E_DALIBridgeCommand.resetDurationTestDoneFlag:
	fbResetDurationTestDoneFlag(
		bStart					:= requestFirstCycle,
		nAddress				:= activeRequest.address,
		eAddressType			:= activeRequest.addressType,
	);
	processResult(
		busy					:= fbResetDurationTestDoneFlag.bBusy,
		bError					:= fbResetDurationTestDoneFlag.bError,
		data					:= 0,
		ipResultMessage			:= fbResetDurationTestDoneFlag.ipResultMessage
	);
	
E_DALIBridgeCommand.resetFunctionTestDoneFlag:
	fbResetFunctionTestDoneFlag(
		bStart					:= requestFirstCycle,
		nAddress				:= activeRequest.address,
		eAddressType			:= activeRequest.addressType,
	);
	processResult(
		busy					:= fbResetFunctionTestDoneFlag.bBusy,
		bError					:= fbResetFunctionTestDoneFlag.bError,
		data					:= 0,
		ipResultMessage			:= fbResetFunctionTestDoneFlag.ipResultMessage
	);
	
E_DALIBridgeCommand.startDurationTest:
	IF emergency THEN
		cancelCommand();
	ELSE
		fbStartDurationTest(
			bStart					:= requestFirstCycle,
			nAddress				:= activeRequest.address,
			eAddressType			:= activeRequest.addressType,
		);
		processResult(
			busy					:= fbStartDurationTest.bBusy,
			bError					:= fbStartDurationTest.bError,
			data					:= 0,
			ipResultMessage			:= fbStartDurationTest.ipResultMessage
		);
	END_IF
	
E_DALIBridgeCommand.startFunctionTest:
	IF emergency THEN
		cancelCommand();
	ELSE
		fbStartFunctionTest(
			bStart					:= requestFirstCycle,
			nAddress				:= activeRequest.address,
			eAddressType			:= activeRequest.addressType,
		);
		processResult(
			busy					:= fbStartFunctionTest.bBusy,
			bError					:= fbStartFunctionTest.bError,
			data					:= 0,
			ipResultMessage			:= fbStartFunctionTest.ipResultMessage
		);
	END_IF
	
E_DALIBridgeCommand.stopTest:
	fbStopTest(
		bStart						:= requestFirstCycle,
		nAddress					:= activeRequest.address,
		eAddressType				:= activeRequest.addressType,
	);
	processResult(
		busy						:= fbStopTest.bBusy,
		bError						:= fbStopTest.bError,
		data						:= 0,
		ipResultMessage				:= fbStopTest.ipResultMessage
	);
	
E_DALIBridgeCommand.setDurationTestInterval:
	fbSetDurationTestInterval(
		bStart						:= requestFirstCycle,
		nAddress					:= activeRequest.address,
		eAddressType				:= activeRequest.addressType,
		nDurationTestInterval		:= activeRequest.data
	);
	processResult(
		busy						:= fbSetDurationTestInterval.bBusy,
		bError						:= fbSetDurationTestInterval.bError,
		data						:= 0,
		ipResultMessage				:= fbSetDurationTestInterval.ipResultMessage
	);
	
E_DALIBridgeCommand.setFunctionTestInterval:
	fbSetFunctionTestInterval(
		bStart						:= requestFirstCycle,
		nAddress					:= activeRequest.address,
		eAddressType				:= activeRequest.addressType,
		nFunctionTestInterval		:= activeRequest.data
	);
	processResult(
		busy						:= fbSetFunctionTestInterval.bBusy,
		bError						:= fbSetFunctionTestInterval.bError,
		data						:= 0,
		ipResultMessage				:= fbSetFunctionTestInterval.ipResultMessage
	);
	
E_DALIBridgeCommand.startIdentification202:
	fbStartIdentification202(
		bStart						:= requestFirstCycle,
		nAddress					:= activeRequest.address,
		eAddressType				:= activeRequest.addressType,
	);
	processResult(
		busy						:= fbStartIdentification202.bBusy,
		bError						:= fbStartIdentification202.bError,
		data						:= 0,
		ipResultMessage				:= fbStartIdentification202.ipResultMessage
	);
	
E_DALIBridgeCommand.queryGroups:
	fbQueryGroups(
		bStart						:= requestFirstCycle,
		nAddress 					:= activeRequest.address,
		eAddressType				:= activeRequest.addressType
	);
	processResult(
		busy						:= fbQueryGroups.bBusy,
		bError						:= fbQueryGroups.bError,
		data						:= fbQueryGroups.nGroups,
		ipResultMessage				:= fbQueryGroups.ipResultMessage
	);
	
E_DALIBridgeCommand.addToGroup:
	fbAddToGroup(
		bStart 						:= requestFirstCycle,
		nAddress 					:= activeRequest.address,
		eAddressType				:= activeRequest.addressType,
		nGroup						:= activeRequest.data
	);
	processResult(
		busy						:= fbAddToGroup.bBusy,
		bError						:= fbAddToGroup.bError,
		data						:= 0,
		ipResultMessage				:= fbAddToGroup.ipResultMessage
	);
	
E_DALIBridgeCommand.removeFromGroup:
	fbRemoveFromGroup(
		bStart						:= requestFirstCycle,
		nAddress 					:= activeRequest.address,
		eAddressType 				:= activeRequest.addressType,
		nGroup						:= activeRequest.data
	);
	processResult(
		busy						:= fbRemoveFromGroup.bBusy,
		bError						:= fbRemoveFromGroup.bError,
		data						:= 0,
		ipResultMessage				:= fbRemoveFromGroup.ipResultMessage
	);
	
E_DALIBridgeCommand.testCommand:
	processResult(
		busy := FALSE,
		data := 123,
		bError := FALSE,
		ipResultMessage := NULL
	);

ELSE
	activeRequest.command := E_DALIBridgeCommand.idle;
END_CASE

processNotifications();

requestFirstCycle := FALSE;

METHOD PRIVATE cancelCommand
VAR_INPUT
END_VAR

VAR
	tmpResponse: ST_DALIBridgeResponse;
END_VAR
// generate response
tmpResponse.valid := TRUE;
tmpResponse.data := 0;
tmpResponse.error := TRUE;
tmpResponse.message := 'Emergency in progress';
tmpResponse.sequence := THIS^.activeRequestSequence;

// return to the idle state, ready for a new request
THIS^.activeRequest.command := E_DALIBridgeCommand.idle;
// publish the response
THIS^.rpcResponse := tmpResponse;
END_METHOD

METHOD FB_init : BOOL
VAR_INPUT
	bInitRetains : BOOL; // if TRUE, the retain variables are initialized (warm start / cold start)
	bInCopyCode : BOOL;  // if TRUE, the instance afterwards gets moved into the copy code (online change)
	
	communication : I_DALICommunication;
END_VAR
THIS^.communication := communication;
END_METHOD

METHOD PRIVATE initCommunication
VAR_INPUT
END_VAR
VAR
	i : INT;
END_VAR
IF communication = 0 THEN
	RETURN;
END_IF

FOR i := 0 TO GVL_DALIBridge.maxInputEventListeners-1 DO
	fbsGetInputNotification[i].ipDALICommunication := communication;
END_FOR

fbEmergencyPowerOn.ipDALICommunication 		:= communication;
fbDirectArcPowerControl.ipDALICommunication := communication;
fbQueryActualLevel.ipDALICommunication 		:= communication;
fbQueryStatus.ipDALICommunication 			:= communication;
fbSetEventScheme.ipDALICommunication 		:= communication;
fbQueryEventScheme.ipDALICommunication 		:= communication;
fbSetEventFilter.ipDALICommunication 		:= communication;
fbQueryEventFilter.ipDALICommunication 		:= communication;
fbIdentifyDevice102.ipDALICommunication 	:= communication;
fbIdentifyDevice103.ipDALICommunication 	:= communication;
fbEnableInstance.ipDALICommunication 		:= communication;
fbGoToScene.ipDALICommunication 			:= communication;
fbSetFadeTime.ipDALICommunication 			:= communication;
fbQueryInputValue.ipDALICommunication		:= communication;

fbQueryBatteryCharge.ipDALICommunication    	:= communication;
fbQueryDurationTestResult.ipDALICommunication 	:= communication;
fbQueryEmergencyMode.ipDALICommunication        := communication;
fbQueryEmergencyStatus.ipDALICommunication  	:= communication;
fbQueryFailureStatus.ipDALICommunication		:= communication;
fbQueryRatedDuration.ipDALICommunication		:= communication;
fbQueryTestTiming.ipDALICommunication			:= communication;
fbResetDurationTestDoneFlag.ipDALICommunication := communication;
fbResetFunctionTestDoneFlag.ipDALICommunication := communication;
fbStartDurationTest.ipDALICommunication 		:= communication;
fbStartFunctionTest.ipDALICommunication 		:= communication;
fbStopTest.ipDALICommunication					:= communication;
fbSetDurationTestInterval.ipDALICommunication   := communication;
fbSetFunctionTestInterval.ipDALICommunication   := communication;
fbStartIdentification202.ipDALICommunication    := communication;
END_METHOD

METHOD PRIVATE isFirstCycle : BOOL
VAR_INPUT
END_VAR
VAR_INST
	fbGetCurTaskIndex : GETCURTASKINDEX;
END_VAR
fbGetCurTaskIndex();
isFirstCycle := TwinCAT_SystemInfoVarList._TaskInfo[fbGetCurTaskIndex.index].FirstCycle;
END_METHOD

METHOD PRIVATE processNotifications : BOOL
VAR_INPUT
END_VAR
VAR
	i 				: DINT;
	eventsProcessed : BYTE := 0;
	
	currentParams   : REFERENCE TO ST_DALIBridgeInputEventParams;
	currentFb 		: REFERENCE TO FB_DALIGetInputNotification;
	currentEvent    : REFERENCE TO ST_DALIBridgeInputEvent;
	
	newNotif : ST_DALIBridgeNotification;
END_VAR
IF NOT notificationAcked THEN
	// cannot process more notifications until the current notification has been ACKed
	processNotifications := FALSE;
	RETURN;
END_IF

newNotif.valid := FALSE;

// for every active notification listener
FOR i := 0 TO numInputEventListeners-1 DO
	IF (eventsProcessed >= GVL_DALIBridge.maxInputEventsPerNotification) THEN
		// stop processing if the event buffer is full
		EXIT;
	END_IF	

	currentFb REF= fbsGetInputNotification[i];
	currentParams REF= inputEventListenerParams[i];
	
	// check for a new event
	currentFb(
		bEnable := TRUE,
		eEventScheme := currentParams.eventScheme,
		nAddressInfo1 := currentParams.addressInfo1,
		nAddressInfo2 := currentParams.addressInfo2
	);
	
	// don't add to event array if no new data was found
	IF NOT currentFb.bNewData THEN
		CONTINUE;
	END_IF
	
	// populate the event entry
	currentEvent REF= newNotif.inputEvents[eventsProcessed];
	currentEvent.data := currentFb.nEventInfo;
	currentEvent.error := currentFb.bError;
	currentFb.ipResultMessage.RequestEventText(
		nLangId := 1033,
		sResult := currentEvent.message,
		nResultSize := SIZEOF(currentEvent.message)
	);
	currentEvent.parameters := inputEventListenerParams[i];
	currentEvent.status := currentFb.ipResultMessage.nEventId;
	
	eventsProcessed := eventsProcessed + 1;
END_FOR

IF (eventsProcessed > 0) THEN
	newNotif.sequence := notificationCounter;
	notificationCounter := notificationCounter + 1;
	newNotif.nInputEvents := eventsProcessed;
	newNotif.valid := TRUE;
	
	notification := newNotif;
	notificationAcked := FALSE;
END_IF
END_METHOD

METHOD PRIVATE processResult
VAR_INPUT
	busy 			: BOOL;
	data            : LWORD;
	bError 			: BOOL;
	ipResultMessage	: Tc3_EventLogger.I_TcMessage;
END_VAR
VAR
	tmpResponse: ST_DALIBridgeResponse;
END_VAR
IF (busy) THEN
	// continue executing the command function block until it is no longer busy
	RETURN;
END_IF

// generate response
tmpResponse.valid := TRUE;
tmpResponse.data := data;
tmpResponse.error := bError;
tmpResponse.sequence := THIS^.activeRequestSequence;
IF ipResultMessage = 0 THEN
	ADSLOGSTR(
		msgCtrlMask := ADSLOG_MSGTYPE_WARN,
		msgFmtStr := 'FB_DALIBridge.processResult: ipResultMessage is null',
		strArg := ''
	);
	tmpResponse.status := 0;
	tmpResponse.message := 'ipResultMessage NULL';
ELSE
	tmpResponse.status := ipResultMessage.nEventId;
	ipResultMessage.RequestEventText(1033, tmpResponse.message, SIZEOF(tmpResponse.message));
END_IF

// return to the idle state, ready for a new request
THIS^.activeRequest.command := E_DALIBridgeCommand.idle;
// publish the response
THIS^.rpcResponse := tmpResponse;
END_METHOD

{attribute 'TcRpcEnable' := '1'}
METHOD PUBLIC RpcAckNotification : BOOL
VAR_INPUT
	// The notification sequence number to acknowledge
	sequence : ULINT;
END_VAR
IF notificationAcked THEN
	// can't acknowledge a notification twice
	RpcAckNotification := FALSE;
	RETURN;
END_IF

IF sequence <> notification.sequence THEN
	// attempt to acknowledge a notification with the wrong sequence number
	RpcAckNotification := FALSE;
	RETURN;
END_IF

RpcAckNotification := TRUE;
notificationAcked := TRUE;
END_METHOD

{attribute 'TcRpcEnable' := '1'}
METHOD PUBLIC RpcAddInputEventListener : BOOL
VAR_INPUT
	parameters : ST_DALIBridgeInputEventParams;
END_VAR
VAR
	i : INT;
END_VAR
ADSLOGSTR(
		msgFmtStr := 'add event listener',
		strArg := '',
		msgCtrlMask := ADSLOG_MSGTYPE_LOG
);

FOR i := 0 TO numInputEventListeners-1 DO
	IF (parameters.eventScheme = inputEventListenerParams[i].eventScheme
		AND parameters.addressInfo1 = inputEventListenerParams[i].addressInfo1
		AND parameters.addressInfo2 = inputEventListenerParams[i].addressInfo2) 
	THEN
		// the desired event listener is already enabled
		RpcAddInputEventListener := TRUE;
		RETURN;
	END_IF
END_FOR

IF numInputEventListeners >= GVL_DALIBridge.maxInputEventListeners THEN
	// notification listeners are full
	RpcAddInputEventListener := FALSE;
	RETURN;
END_IF

inputEventListenerParams[numInputEventListeners] := parameters;
numInputEventListeners := numInputEventListeners + 1;

RpcAddInputEventListener := TRUE;
END_METHOD

{attribute 'TcRpcEnable' := '1'}
METHOD PUBLIC RpcHandshake
VAR_INPUT
END_VAR
VAR_OUTPUT
	protocolVersion : INT;
END_VAR
protocolVersion := 2;
END_METHOD

(* Called by an external API consumer over RPC to start a DALI request.
   Returns TRUE if the request was accepted. If the bridge is busy, then this returns FALSE
   and the request will not be processed. *)
{attribute 'TcRpcEnable' := '1'}
METHOD PUBLIC RpcRequest : BOOL
VAR_INPUT
	// The DALI operation that the caller wants the DALI Bridge to perform.
	request : ST_DALIBridgeRequest;
END_VAR
VAR_OUTPUT
	// A sequence number that will allow the caller to identify the response value.
	sequence : ULINT;
END_VAR
// reject request if bridge is busy processing a previous request
IF (THIS^.activeRequest.command <> E_DALIBridgeCommand.idle) THEN
	RpcRequest := FALSE;
	RETURN;
END_IF

// save the request, so it will begin processing next cycle
THIS^.activeRequest := request;
THIS^.activeRequestSequence := THIS^.requestCounter;
sequence := THIS^.activeRequestSequence;

// advance sequence counter
THIS^.requestCounter := THIS^.requestCounter + 1;

// The next cycle will be the first cycle of the new request
THIS^.requestFirstCycle := TRUE;

RpcRequest := TRUE;
END_METHOD

{attribute 'TcRpcEnable' := '1'}
METHOD PUBLIC RpcReset
VAR_INPUT
END_VAR
numInputEventListeners := 0;
notificationAcked := TRUE;
activeRequest.command := E_DALIBridgeCommand.idle;
ADSLOGSTR(
		msgFmtStr := 'reset FB_DALIBridge',
		strArg := '',
		msgCtrlMask := ADSLOG_MSGTYPE_LOG
);
END_METHOD

END_FUNCTION_BLOCK

// ---- GlobalTextList.TcGTLO
TEXTLIST GlobalTextList
  621 = '%d'
  665 = '%d %'
  2025 = '%d ms'
  1540 = '%d s'
  646 = '%s'
  640 = '0'
  641 = '1'
  661 = '10'
  662 = '11'
  663 = '12'
  999 = '13'
  1000 = '14'
  1001 = '15'
  1002 = '16'
  1003 = '17'
  1004 = '18'
  1005 = '19'
  642 = '2'
  1006 = '20'
  1007 = '21'
  1008 = '22'
  1009 = '23'
  1010 = '24'
  1011 = '25'
  1012 = '26'
  1013 = '27'
  1014 = '28'
  1015 = '29'
  654 = '3'
  1016 = '30'
  1017 = '31'
  1018 = '32'
  1019 = '33'
  1020 = '34'
  1021 = '35'
  1022 = '36'
  1023 = '37'
  1024 = '38'
  1025 = '39'
  655 = '4'
  1026 = '40'
  1027 = '41'
  1028 = '42'
  1029 = '43'
  1030 = '44'
  1031 = '45'
  1032 = '46'
  1033 = '47'
  1034 = '48'
  1035 = '49'
  656 = '5'
  358 = '50'
  359 = '51'
  360 = '52'
  361 = '53'
  362 = '54'
  363 = '55'
  364 = '56'
  365 = '57'
  366 = '58'
  367 = '59'
  657 = '6'
  368 = '60'
  369 = '61'
  370 = '62'
  371 = '63'
  658 = '7'
  659 = '8'
  660 = '9'
  1089 = 'AC-supply possible'
  644 = 'Actual Level:'
  650 = 'Address Type'
  1175 = 'AM Operation active:'
  1044 = 'AM operation possible'
  2131 = 'Back'
  2471 = 'Bit 0'
  379 = 'Bit 1'
  2734 = 'Bit 2'
  2320 = 'Bit 3'
  929 = 'Bit 4'
  2576 = 'Bit 5'
  2065 = 'Bit 6'
  1623 = 'Bit 7'
  626 = 'Broadcast'
  515 = 'Button pressed'
  498 = 'Button released'
  527 = 'Button stuck / free'
  593 = 'Cancel Hold Timer'
  2101 = 'Catch Movement'
  2319 = 'Catching:'
  897 = 'Change Addresses'
  372 = 'Choose group:'
  98 = 'Choose scene:'
  618 = 'Complete new installation \n(all addresses will be removed)'
  807 = 'Control'
  645 = 'Control Gear Failure:'
  146 = 'Control LED'
  445 = 'Current protection active:'
  1716 = 'Current protection device'
  668 = 'Current protection enabled:'
  5 = 'Current Protector Enabled '
  1902 = 'DALI Line:'
  1135 = 'DC-supply possible'
  560 = 'Deadtime Timer:'
  1180 = 'DI1 falling edge'
  1218 = 'DI1 rising edge'
  1726 = 'DI2 falling edge'
  1876 = 'DI2 rising edge'
  936 = 'Dimming Curve:'
  2135 = 'Do not lock process image in case of \nDALI commands from DI1 or DI2'
  519 = 'Double press'
  1112 = 'Double Timer Min:'
  482 = 'Double Timer:'
  811 = 'Down'
  486 = 'Enable'
  828 = 'Enable:'
  1982 = 'EventPriority'
  32 = 'EventPriority:'
  1925 = 'EventScheme'
  1113 = 'EventScheme:'
  1841 = 'Extended Fade Time only valid if Fade Time equals 0!'
  310 = 'Extended Version Number'
  649 = 'Fade Running:'
  494 = 'FadeRate'
  499 = 'FadeTime'
  319 = 'Fast Fade Time:'
  1808 = 'Features LED'
  1434 = 'GearType LED'
  815 = 'Go to Scene'
  99 = 'Go to scene'
  625 = 'Group Address'
  568 = 'Hold Timer:'
  311 = 'Hysteresis Min:'
  313 = 'Hysteresis:'
  1117 = 'Identify'
  315 = 'Illuminance Level'
  540 = 'Input Value:'
  544 = 'Instance Error:'
  1038 = 'Instance Number:'
  492 = 'Internal DALI power supply disabled'
  1771 = 'K-Bus Watchdog'
  647 = 'Lamp Failure:'
  506 = 'LED module integrated'
  306 = 'Load Decrease:'
  1137 = 'Load Increase:'
  1811 = 'Lockable bytes: changeable if "Offset 2" has the Value 85 (0x55).\nFor changing use decimal value.'
  1077 = 'Login'
  1294 = 'Logout'
  523 = 'Long press repeat'
  507 = 'Long press start'
  511 = 'Long press stop'
  2046 = 'Memory Bank:'
  584 = 'Movement'
  531 = 'na'
  680 = 'Name'
  926 = 'Name of byte in memory bank'
  56 = 'NewAddress'
  588 = 'No Movement'
  2294 = 'None'
  572 = 'Occupied'
  808 = 'Off'
  674 = 'Offset'
  1329 = 'Offset in memory bank'
  55 = 'OldAddress'
  816 = 'On and Step Up'
  277 = 'Open Circuit:'
  1714 = 'Operator'
  619 = 'Optical feedback'
  963 = 'Output is current controlled'
  826 = 'Output regulated by current:'
  1900 = 'Parameters'
  2547 = 'Parameters Absolute Input Device'
  1580 = 'Parameters Generic Instance'
  309 = 'Parameters Light Sensor'
  556 = 'Parameters Occupancy Sensor'
  465 = 'Parameters Pushbutton Sensor'
  1847 = 'Physical selection supported'
  1071 = 'Please check if Current Protector is present \nby reading parameters first.'
  308 = 'Please select the desired Short Address in the table above.'
  751 = 'Position Event'
  930 = 'Possible Operating Modes LED'
  719 = 'Power pulse operation'
  1744 = 'Power supply integrated'
  1561 = 'PP Operation active:'
  970 = 'PWM Operation active:'
  1882 = 'PWM operation possible'
  1487 = 'Query idle time detection \nenabled'
  701 = 'Query load decrease enabled'
  1351 = 'Query load increase enabled'
  837 = 'Query reduction luminous flux \nregarding thermal overload'
  463 = 'Query short circuit enabled'
  1293 = 'Query thermal switch enabled'
  617 = 'Random Addressing'
  373 = 'Read'
  181 = 'Read Parameters'
  1531 = 'Reads all Fading Parameters'
  810 = 'Recall Max Level'
  809 = 'Recall Min Level'
  186 = 'Ref. Measurement failed:'
  439 = 'Reference System Power'
  580 = 'Repeat'
  470 = 'Repeat Timer:'
  564 = 'Report Timer:'
  2418 = 'Reset inactive process image'
  648 = 'Reset State:'
  1037 = 'Resolution:'
  616 = 'Scan devices by address'
  1036 = 'Scene Level'
  814 = 'Scene:'
  1366 = 'Set Extended Fade Time'
  252 = 'Set Fade Rate'
  1875 = 'Set Fade Time'
  624 = 'Short Address'
  302 = 'Short Address Range'
  1041 = 'Short Address:'
  34 = 'Short Circuit:'
  503 = 'Short press'
  1516 = 'Short Timer Min:'
  478 = 'Short Timer:'
  300 = 'Single Short Address'
  615 = 'Start'
  620 = 'Start with address:'
  643 = 'Status'
  958 = 'Status Absolute Input Device'
  2506 = 'Status Generic Instance'
  82 = 'Status LED'
  317 = 'Status Light Sensor'
  597 = 'Status Occupancy Sensor'
  536 = 'Status Pushbutton Sensor'
  812 = 'Step Down'
  813 = 'Step Down and Off'
  818 = 'Step Up'
  164 = 'Stuck Timer:'
  376 = 'Switch Off'
  375 = 'Switch On'
  2458 = 'Terminal Event'
  1108 = 'Thermal Overload:'
  355 = 'Thermal Shut Down:'
  305 = 'To'
  627 = 'Unaddressed'
  817 = 'Up'
  2521 = 'V%s'
  576 = 'Vacant'
  1205 = 'Value'
  686 = 'Value Dec'
  1435 = 'Value decimal'
  692 = 'Value Hex'
  2231 = 'Value hexadecimal,\nto change use\nvalue decimal'
  374 = 'Write'
  1047 = 'Write default values'
  490 = 'Write parameters'
END_TEXTLIST

// ---- Tc3_DALI_PLC_Commissioning_Tool/GlobalTextList_1.TcGTLO
TEXTLIST GlobalTextList_1
  621 = '%d'
  665 = '%d %'
  2025 = '%d ms'
  1540 = '%d s'
  646 = '%s'
  640 = '0'
  641 = '1'
  661 = '10'
  662 = '11'
  663 = '12'
  999 = '13'
  1000 = '14'
  1001 = '15'
  1002 = '16'
  1003 = '17'
  1004 = '18'
  1005 = '19'
  642 = '2'
  1006 = '20'
  1007 = '21'
  1008 = '22'
  1009 = '23'
  1010 = '24'
  1011 = '25'
  1012 = '26'
  1013 = '27'
  1014 = '28'
  1015 = '29'
  654 = '3'
  1016 = '30'
  1017 = '31'
  1018 = '32'
  1019 = '33'
  1020 = '34'
  1021 = '35'
  1022 = '36'
  1023 = '37'
  1024 = '38'
  1025 = '39'
  655 = '4'
  1026 = '40'
  1027 = '41'
  1028 = '42'
  1029 = '43'
  1030 = '44'
  1031 = '45'
  1032 = '46'
  1033 = '47'
  1034 = '48'
  1035 = '49'
  656 = '5'
  358 = '50'
  359 = '51'
  360 = '52'
  361 = '53'
  362 = '54'
  363 = '55'
  364 = '56'
  365 = '57'
  366 = '58'
  367 = '59'
  657 = '6'
  368 = '60'
  369 = '61'
  370 = '62'
  371 = '63'
  658 = '7'
  659 = '8'
  660 = '9'
  1089 = 'AC-supply possible'
  644 = 'Actual Level:'
  650 = 'Address Type'
  1175 = 'AM Operation active:'
  1044 = 'AM operation possible'
  2131 = 'Back'
  2471 = 'Bit 0'
  379 = 'Bit 1'
  2734 = 'Bit 2'
  2320 = 'Bit 3'
  929 = 'Bit 4'
  2576 = 'Bit 5'
  2065 = 'Bit 6'
  1623 = 'Bit 7'
  803 = 'Broadcast'
  515 = 'Button pressed'
  498 = 'Button released'
  527 = 'Button stuck / free'
  593 = 'Cancel Hold Timer'
  2101 = 'Catch Movement'
  2319 = 'Catching:'
  897 = 'Change Addresses'
  372 = 'Choose group:'
  98 = 'Choose scene:'
  618 = 'Complete new installation \n(all addresses will be removed)'
  807 = 'Control'
  645 = 'Control Gear Failure:'
  146 = 'Control LED'
  445 = 'Current protection active:'
  1716 = 'Current protection device'
  668 = 'Current protection enabled:'
  5 = 'Current Protector Enabled '
  1902 = 'DALI Line:'
  334 = 'DALI Power Supply'
  1135 = 'DC-supply possible'
  560 = 'Deadtime Timer:'
  1180 = 'DI1 falling edge'
  1218 = 'DI1 rising edge'
  1726 = 'DI2 falling edge'
  1876 = 'DI2 rising edge'
  936 = 'Dimming Curve:'
  169 = 'Do not lock process image'
  2135 = 'Do not lock process image in case of \nDALI commands from DI1 or DI2'
  2344 = 'Do not lock process image in case of DALI commands from DI1 or DI2'
  519 = 'Double press'
  1112 = 'Double Timer Min:'
  482 = 'Double Timer:'
  811 = 'Down'
  486 = 'Enable'
  828 = 'Enable:'
  1982 = 'EventPriority'
  32 = 'EventPriority:'
  494 = 'EventScheme'
  1113 = 'EventScheme:'
  1841 = 'Extended Fade Time only valid if Fade Time equals 0!'
  310 = 'Extended Version Number'
  649 = 'Fade Running:'
  1150 = 'FadeRate'
  1160 = 'FadeTime'
  319 = 'Fast Fade Time:'
  1808 = 'Features LED'
  1434 = 'GearType LED'
  815 = 'Go to Scene'
  99 = 'Go to scene'
  802 = 'Group Address'
  1923 = 'Hier noch die Abfrage der extended version Number\nmit reinbringen, damit klar wird welcher Edition das Gerät angehört.'
  568 = 'Hold Timer:'
  311 = 'Hysteresis Min:'
  313 = 'Hysteresis:'
  1117 = 'Identify'
  2159 = 'Identify 202'
  315 = 'Illuminance Level'
  540 = 'Input Value:'
  544 = 'Instance Error:'
  1038 = 'Instance Number:'
  1374 = 'InstanceType0'
  652 = 'InstanceType1'
  653 = 'InstanceType3'
  664 = 'InstanceType4'
  492 = 'Internal DALI power supply disabled'
  1820 = 'IT0 (Generic Input)'
  1151 = 'IT1 (PushButton)'
  906 = 'IT2 (absolute Input)'
  909 = 'IT2 (Absolute Input)'
  819 = 'IT3 (Occupancy)'
  224 = 'IT4 (Light Sensor)'
  1771 = 'K-Bus Watchdog'
  647 = 'Lamp Failure:'
  506 = 'LED module integrated'
  306 = 'Load Decrease:'
  1137 = 'Load Increase:'
  1811 = 'Lockable bytes: changeable if "Offset 2" has the Value 85 (0x55).\nFor changing use decimal value.'
  523 = 'Long press repeat'
  507 = 'Long press start'
  511 = 'Long press stop'
  2046 = 'Memory Bank:'
  584 = 'Movement'
  531 = 'na'
  842 = 'Name'
  926 = 'Name of byte in memory bank'
  193 = 'NewAddress'
  588 = 'No Movement'
  572 = 'Occupied'
  808 = 'Off'
  835 = 'Offset'
  1329 = 'Offset in memory bank'
  192 = 'OldAddress'
  816 = 'On and Step Up'
  277 = 'Open Circuit:'
  651 = 'OperatingMode'
  619 = 'Optical feedback'
  963 = 'Output is current controlled'
  826 = 'Output regulated by current:'
  1900 = 'Parameters'
  2547 = 'Parameters Absolute Input Device'
  1580 = 'Parameters Generic Instance'
  309 = 'Parameters Light Sensor'
  556 = 'Parameters Occupancy Sensor'
  465 = 'Parameters Pushbutton Sensor'
  1847 = 'Physical selection supported'
  1071 = 'Please check if Current Protector is present \nby reading parameters first.'
  308 = 'Please select the desired Short Address in the table above.'
  751 = 'Position Event'
  930 = 'Possible Operating Modes LED'
  719 = 'Power pulse operation'
  1744 = 'Power supply integrated'
  1561 = 'PP Operation active:'
  970 = 'PWM Operation active:'
  1882 = 'PWM operation possible'
  1487 = 'Query idle time detection \nenabled'
  701 = 'Query load decrease enabled'
  1351 = 'Query load increase enabled'
  837 = 'Query reduction luminous flux \nregarding thermal overload'
  463 = 'Query short circuit enabled'
  1293 = 'Query thermal switch enabled'
  617 = 'Random Addressing'
  373 = 'Read'
  316 = 'Read parameters'
  181 = 'Read Parameters'
  1531 = 'Reads all Fading Parameters'
  810 = 'Recall Max Level'
  809 = 'Recall Min Level'
  186 = 'Ref. Measurement failed:'
  439 = 'Reference System Power'
  580 = 'Repeat'
  470 = 'Repeat Timer:'
  564 = 'Report Timer:'
  2418 = 'Reset inactive process image'
  648 = 'Reset State:'
  1037 = 'Resolution:'
  616 = 'Scan devices by address'
  1036 = 'Scene Level'
  814 = 'Scene:'
  1366 = 'Set Extended Fade Time'
  252 = 'Set Fade Rate'
  1875 = 'Set Fade Time'
  801 = 'Short Address'
  1179 = 'Short Address Range'
  1041 = 'Short Address:'
  34 = 'Short Circuit:'
  503 = 'Short press'
  1516 = 'Short Timer Min:'
  478 = 'Short Timer:'
  1170 = 'Single Short Address'
  615 = 'Start'
  620 = 'Start with address:'
  643 = 'Status'
  958 = 'Status Absolute Input Device'
  2506 = 'Status Generic Instance'
  82 = 'Status LED'
  317 = 'Status Light Sensor'
  597 = 'Status Occupancy Sensor'
  536 = 'Status Pushbutton Sensor'
  812 = 'Step Down'
  813 = 'Step Down and Off'
  818 = 'Step Up'
  164 = 'Stuck Timer:'
  376 = 'Switch Off'
  375 = 'Switch On'
  2458 = 'Terminal Event'
  1108 = 'Thermal Overload:'
  355 = 'Thermal Shut Down:'
  305 = 'To'
  804 = 'Unaddressed'
  817 = 'Up'
  2521 = 'V%s'
  298 = 'V3.1.1.0'
  858 = 'V3.4.0.0'
  395 = 'V3.4.0.1'
  1169 = 'V3.5.0.0'
  576 = 'Vacant'
  1205 = 'Value'
  850 = 'Value Dec'
  1435 = 'Value decimal'
  857 = 'Value Hex'
  2231 = 'Value hexadecimal,\nto change use\nvalue decimal'
  374 = 'Write'
  1047 = 'Write default values'
  490 = 'Write parameters'
END_TEXTLIST

// ---- Tc3_DALI_PLC_Commissioning_Tool/VISUs/TextLists/CommandOnTerminalEvent.TcTLO
TEXTLIST CommandOnTerminalEvent
  0 = 'Do Nothing'
  1 = 'Off'
  2 = 'RecallMaxLevel'
  3 = 'RecallMinLevel'
  4 = 'GoToScene0'
  5 = 'GoToScene1'
  6 = 'GoToScene2'
  7 = 'GoToScene3'
  8 = 'GoToScene4'
  9 = 'GoToScene5'
  10 = 'GoToScene6'
  11 = 'GoToScene7'
  12 = 'GoToScene8'
  13 = 'GoToScene9'
  14 = 'GoToScene10'
  15 = 'GoToScene11'
  16 = 'GoToScene12'
  17 = 'GoToScene13'
  18 = 'GoToScene14'
  19 = 'GoToScene15'
   = ''
END_TEXTLIST

// ---- Tc3_DALI_PLC_Commissioning_Tool/VISUs/TextLists/DimmingCurve.TcTLO
TEXTLIST DimmingCurve
  0 = 'Logarithmic'
  1 = 'Linear'
  255 = 'Unknown'
   = ''
END_TEXTLIST

// ---- Tc3_DALI_PLC_Commissioning_Tool/VISUs/TextLists/EventPriority.TcTLO
TEXTLIST EventPriority
  2 = 'MiddleHigh'
  3 = 'Middle'
  4 = 'MiddleLow'
  5 = 'Low'
  255 = 'Unknown'
   = ''
END_TEXTLIST

// ---- Tc3_DALI_PLC_Commissioning_Tool/VISUs/TextLists/EventScheme.TcTLO
TEXTLIST EventScheme
  0 = '0 - Instance type and number'
  1 = '1 - Short address and instance type'
  2 = '2 - Short address and instance number'
  3 = '3 - Device group and instance type'
  4 = '4 - Instance group and instance type'
   = ''
END_TEXTLIST

// ---- Tc3_DALI_PLC_Commissioning_Tool/VISUs/TextLists/ExtendedFadeTime.TcTLO
TEXTLIST ExtendedFadeTime
  0 = 'No Fade'
  1 = '1 * 100 ms = 100 ms'
  2 = '2 * 100 ms = 200 ms'
  3 = '3 * 100 ms = 300 ms'
  4 = '4 * 100 ms = 400 ms'
  5 = '5 * 100 ms = 500 ms'
  6 = '6 * 100 ms = 600 ms'
  7 = '7 * 100 ms = 700 ms'
  8 = '8 * 100 ms = 800 ms'
  9 = '9 * 100 ms = 900 ms'
  10 = '10 * 100 ms = 1000 ms'
  11 = '11 * 100 ms = 1100 ms'
  12 = '12 * 100 ms = 1200 ms'
  13 = '13 * 100 ms = 1300 ms'
  14 = '14 * 100 ms = 1400 ms'
  15 = '15 * 100 ms = 1500 ms'
  16 = '16 * 100 ms = 1600 ms'
  17 = '1 * 1 s = 1 s'
  18 = '2 * 1 s = 2 s'
  19 = '3 * 1 s = 3 s'
  20 = '4 * 1 s = 4 s'
  21 = '5 * 1 s = 5 s'
  22 = '6 * 1 s = 6 s'
  23 = '7 * 1 s = 7 s'
  24 = '8 * 1 s = 8 s'
  25 = '9 * 1 s = 9 s'
  26 = '10 * 1 s = 10 s'
  27 = '11 * 1 s = 11 s'
  28 = '12 * 1 s = 12 s'
  29 = '13 * 1 s = 13 s'
  30 = '14 * 1 s = 14 s'
  31 = '15 * 1 s = 15 s'
  32 = '16 * 1 s = 16 s'
  33 = '1 * 10 s = 10 s'
  34 = '2 * 10 s = 20 s'
  35 = '3 * 10 s = 30 s'
  36 = '4 * 10 s = 40 s'
  37 = '5 * 10 s = 50 s'
  38 = '6 * 10 s = 60 s'
  39 = '7 * 10 s = 70 s'
  40 = '8 * 10 s = 80 s'
  41 = '9 * 10 s = 90 s'
  42 = '10 * 10 s = 100 s'
  43 = '11 * 10 s = 110 s'
  44 = '12 * 10 s = 120 s'
  45 = '13 * 10 s = 130 s'
  46 = '14 * 10 s = 140 s'
  47 = '15 * 10 s = 150 s'
  48 = '16 * 10 s = 160 s'
  49 = '1 * 1 min = 1 min'
  50 = '2 * 1 min = 2 min'
  51 = '3 * 1 min = 3 min'
  52 = '4 * 1 min = 4 min'
  53 = '5 * 1 min = 5 min'
  54 = '6 * 1 min = 6 min'
  55 = '7 * 1 min = 7 min'
  56 = '8 * 1 min = 8 min'
  57 = '9 * 1 min = 9 min'
  58 = '10 * 1 min = 10 min'
  59 = '11 * 1 min = 11 min'
  60 = '12 * 1 min = 12 min'
  61 = '13 * 1 min = 13 min'
  62 = '14 * 1 min = 14 min'
  63 = '15 * 1 min = 15 min'
  64 = '16 * 1 min = 16 min'
  255 = 'Unknown'
   = ''
END_TEXTLIST

// ---- Tc3_DALI_PLC_Commissioning_Tool/VISUs/TextLists/FadeRate.TcTLO
TEXTLIST FadeRate
  0 = 'Unknown'
  1 = '358 steps/s'
  2 = '253 steps/s'
  3 = '179 steps/s'
  4 = '127 steps/s'
  5 = '89,4 steps/s'
  6 = '63,3 steps/s'
  7 = '44,7 steps/s'
  8 = '31,6 steps/s'
  9 = '22,4 steps/s'
  10 = '15,8 steps/s'
  11 = '11,2 steps/s'
  12 = '7,9 steps/s'
  13 = '5,6 steps/s'
  14 = '4,0 steps/s'
  15 = '2,8 steps/s'
  255 = 'Unknown'
   = ''
END_TEXTLIST

// ---- Tc3_DALI_PLC_Commissioning_Tool/VISUs/TextLists/FadeTime.TcTLO
TEXTLIST FadeTime
  0 = 'Extended Fade Time'
  1 = '0,7 s'
  2 = '1,0 s'
  3 = '1,4 s'
  4 = '2,0 s'
  5 = '2,8 s'
  6 = '4,0 s'
  7 = '5,7 s'
  8 = '8,0 s'
  9 = '11,3 s'
  10 = '16,0 s'
  11 = '22,6 s'
  12 = '32,0 s'
  13 = '45,3 s'
  14 = '64,0 s'
  15 = '90,5 s'
   = ''
END_TEXTLIST

// ---- Tc3_DALI_PLC_Commissioning_Tool/VISUs/TextLists/FastFadeTime.TcTLO
TEXTLIST FastFadeTime
  0 = 'Disabled'
  4 = 'T100ms'
  8 = 'T200ms'
  12 = 'T300ms'
  16 = 'T400ms'
  20 = 'T500ms'
  24 = 'T600ms'
  27 = 'T700ms'
  255 = 'Unknown'
   = ''
END_TEXTLIST

// ---- Tc3_DALI_PLC_Commissioning_Tool/VISUs/TextLists/TextList_Dialogs.TcTLO
TEXTLIST TextList_Dialogs
  0 = 'Control Gears - Commands'
  1 = 'Control Gears - Parameters'
  2 = 'Control Gears - Addressing'
  3 = 'Control Gears - Groups'
  4 = 'Control Gears - Scenes'
  5 = 'Control Gears - Memory Pages'
  6 = 'Control Gears - Set Fading'
  7 = 'Control Gears - Device Type 6 (LED)'
  8 = 'Control Devices - Parameters'
  9 = 'Control Devices - Addressing'
  10 = 'Control Devices - Device Type 1 (Push button)'
  11 = 'Control Devices - Device Type 2 (Absolute input)'
  12 = 'Control Devices - Device Type 3 (Occupancy sensor)'
  13 = 'Control Devices - Device Type 4 (Light sensor)'
  14 = 'Control Devices - Device Type 0 (Generic instance)'
  15 = 'Control Devices - Memory Pages'
  16 = 'Options KL6821'
   = ''
END_TEXTLIST

// ---- Tc3_DALI_PLC_Commissioning_Tool/VISUs/Visu_DALICommissioning.TcVIS
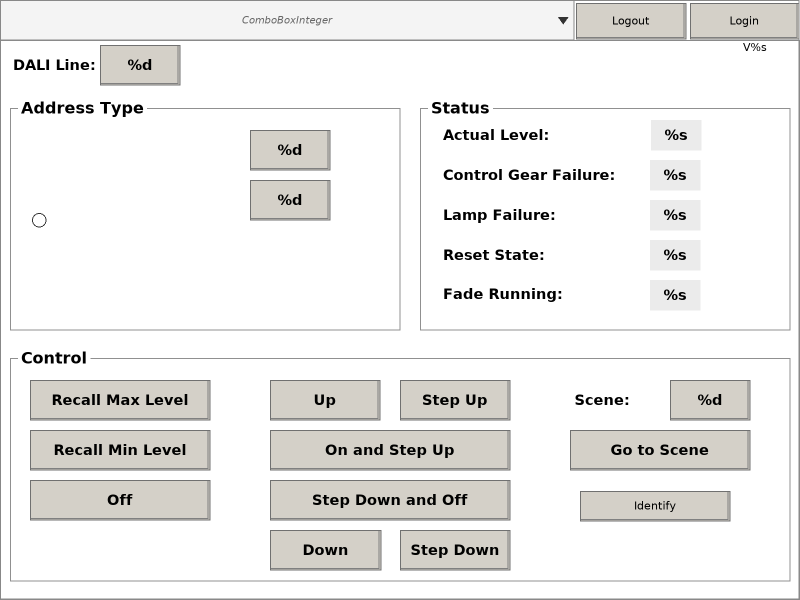
VISUALIZATION Visu_DALICommissioning  // 800x600
    ComboBoxInteger (0,0 574x40), variable: DALI_Commissioning.nSelectedDialog, input disabled if: DALI_Commissioning.bDisableComboBox, text list: 'TextList_Dialogs'
    Frame (0,40 800x560), frame switch variable: DALI_Commissioning.nSelectedDialog
        shows Visu_Part102Commands()
        shows Visu_Part102Parameters()
        shows Visu_Part102Addressing()
        shows Visu_Part102Groups()
        shows Visu_Part102Scenes()
        shows Visu_Part102MemoryBank()
        shows Visu_Part102SetFading()
        shows Visu_Part207Status()
        shows Visu_Part103Parameters()
        shows Visu_Part103Addressing()
        shows Visu_Part301PushButton()
        shows Visu_Part302AbsoluteInputDevice()
        shows Visu_Part303OccupancySensor()
        shows Visu_Part304LightSensor()
        shows Visu_Part300GenericDevice()
        shows Visu_Part103MemoryBank()
        shows Visu_KL6821Configuration()
    Button (690,3 109x36), "Login"
        OnMouseClick: VisuUserMgmt Type=Login
    Button (576,3 110x36), "Logout"
        OnMouseClick: VisuUserMgmt Type=Logout
END_VISUALIZATION

// ---- Tc3_DALI_PLC_Commissioning_Tool/VISUs/Visu_DALICommissioning/Visu_KL6821Configuration.TcVIS
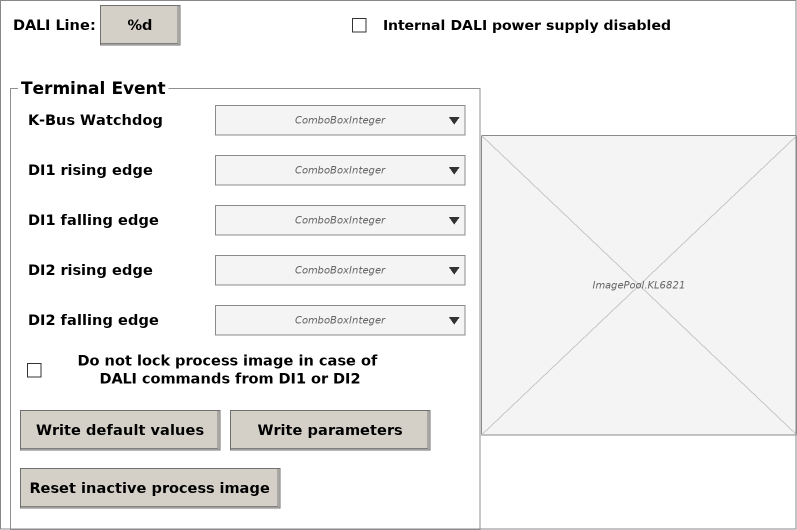
VISUALIZATION Visu_KL6821Configuration  // 797x530
    GroupBox (10,80 470x450), "Terminal Event"
        Textfield (15,25 170x30), "K-Bus Watchdog"
        ComboBoxInteger (205,25 250x30), variable: Communication.eCommandKBusWatchdog, text list: 'CommandOnTerminalEvent'
        Textfield (15,75 170x30), "DI1 rising edge"
        Textfield (15,125 170x30), "DI1 falling edge"
        ComboBoxInteger (205,75 250x30), variable: Communication.eCommandDI1RisingEdge, text list: 'CommandOnTerminalEvent'
        ComboBoxInteger (205,125 250x30), variable: Communication.eCommandDI1FallingEdge, text list: 'CommandOnTerminalEvent'
        Textfield (15,175 170x30), "DI2 rising edge"
        ComboBoxInteger (205,175 250x30), variable: Communication.eCommandDI2RisingEdge, text list: 'CommandOnTerminalEvent'
        Textfield (15,225 170x30), "DI2 falling edge"
        ComboBoxInteger (205,225 250x30), variable: Communication.eCommandDI2FallingEdge, text list: 'CommandOnTerminalEvent'
        Button (220,330 200x40), "Write parameters"
            OnMouseClick: execute { Communication.bInitialize := TRUE; }
        Button (10,330 200x40), "Write default values"
            OnMouseClick: execute { Communication.bDefaultValues := TRUE; }
        Button (10,388 260x40), "Reset inactive process image"
            OnMouseClick: execute { Communication.bResetInactiveProcessImage := TRUE; }
        Checkbox (15,275 35x30), variable: Communication.bDoNotLockProcessImage
        Textfield (50,267 340x45), "Do not lock process image in case of DALI commands from DI1 or DI2"
    Image (481,135 316x300), image: ImagePool.KL6821
    Group (350,10 330x30)
        Checkbox (0,0 34x30), variable: Communication.bInternalPowerSupplyDisabled
        Textfield (30,0 294x30), "Internal DALI power supply disabled"
    Group (10,5 170x40)
        Textfield (0,0 110x40), "DALI Line:"
        Button (90,0 80x40), "%d", text variable: GVL_Internal.nDALILine
            OnMouseClick: write the text variable via Default, min 1, max GVL_Internal.nNumberOfDALI_Lines, title "Choose line"
END_VISUALIZATION

// ---- Tc3_DALI_PLC_Commissioning_Tool/VISUs/Visu_DALICommissioning/Visu_Part102Addressing.TcVIS
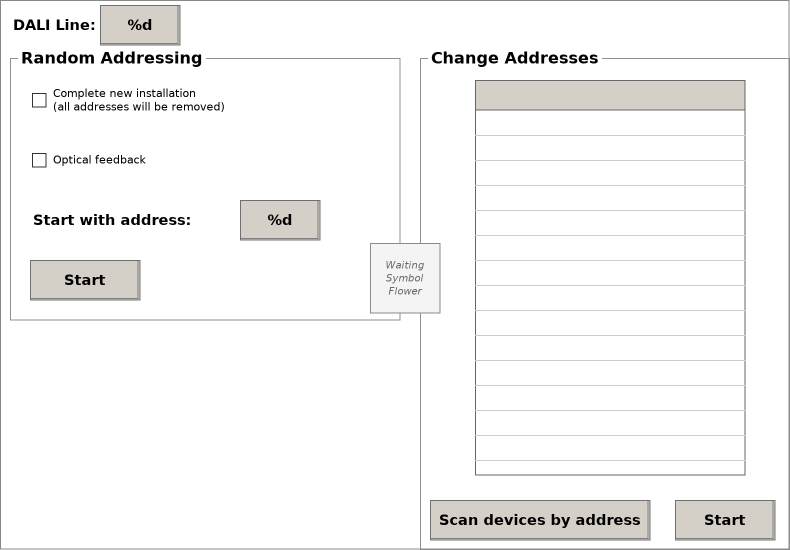
VISUALIZATION Visu_Part102Addressing  // 790x550
    GroupBox (420,50 370x500), "Change Addresses"
        Table (55,30 270x395), data array: DALI_Commissioning.fbPart102Addressing.aChangeAddressList
            p3854506369: DALI_Commissioning.fbPart102Addressing.aChangeAddressList[INDEX].nOldAddress
            p1892666644: DALI_Commissioning.fbPart102Addressing.aChangeAddressList[INDEX].nNewAddress
            p338671338: DALI_Commissioning.fbPart102Addressing.aChangeAddressList[INDEX].nRandomAddress
            p2170511999: DALI_Commissioning.fbPart102Addressing.aChangeAddressList[INDEX].nErrors
            Columns.Column.[0].Template: DALI_Commissioning.fbPart102Addressing.aNoShortAddress[INDEX]
            Columns.Column.[1].Template: DALI_Commissioning.fbPart102Addressing.aNoShortAddress[INDEX]; OnMouseClick: write the text variable via Default, min 0, max 63, title "New Short Address"
        Button (255,450 100x40), "Start"
            OnMouseClick: execute { DALI_Commissioning.fbPart102Addressing.bStartChangeAddress := TRUE; }
        Button (10,450 220x40), "Scan devices by address"
            OnMouseClick: execute { DALI_Commissioning.fbPart102Addressing.bScanDevices := TRUE; }
    GroupBox (10,50 390x270), "Random Addressing"
        Button (20,210 110x40), "Start"
            OnMouseClick: execute { DALI_Commissioning.fbPart102Addressing.bStartRandomAddressing := TRUE; }
        Checkbox (20,30 360x40), "Complete new installation (all addresses will be removed)", variable: DALI_Commissioning.fbPart102Addressing.bNewInstallation
        Checkbox (20,90 360x40), "Optical feedback", variable: DALI_Commissioning.fbPart102Addressing.bOpticalFeedback
        Textfield (20,150 200x40), "Start with address:"
        Button (230,150 80x40), "%d", text variable: DALI_Commissioning.fbPart102Addressing.nStartAddress
            OnMouseClick: write the text variable via Default, min 0, max 63, title "Insert Short Address"
    WaitingSymbolFlower (370,243 70x70), invisible if: DALI_Commissioning.fbPart102Addressing.bHideWaitSymbol
    Group (10,5 170x40)
        Textfield (0,0 110x40), "DALI Line:"
        Button (90,0 80x40), "%d", text variable: GVL_Internal.nDALILine
            OnMouseClick: write the text variable via Default, min 1, max GVL_Internal.nNumberOfDALI_Lines, title "Choose line"
END_VISUALIZATION

// ---- Tc3_DALI_PLC_Commissioning_Tool/VISUs/Visu_DALICommissioning/Visu_Part102Commands.TcVIS
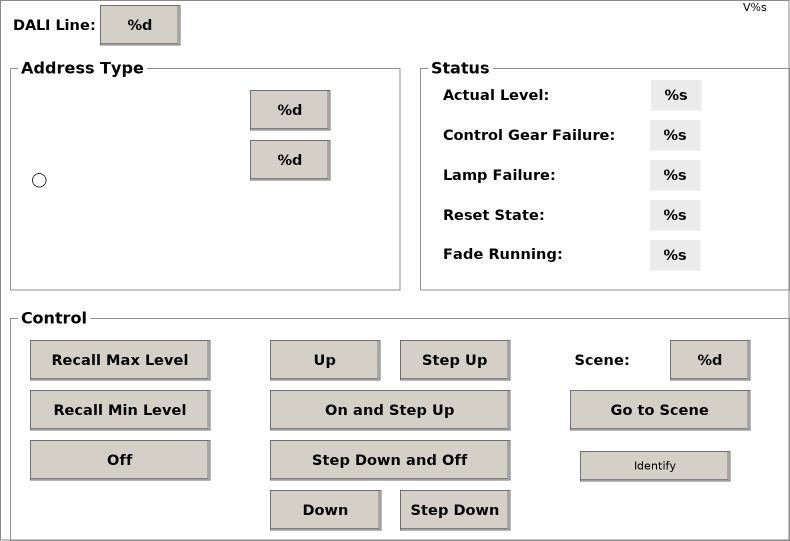
VISUALIZATION Visu_Part102Commands  // 790x541
    GroupBox (10,310 780x231), "Control"
        Button (20,130 180x40), "Off"
            OnMouseClick: execute { DALI_Commissioning.fbPart102Commands.bOff := TRUE; }
        Button (20,80 180x40), "Recall Min Level"
            OnMouseClick: execute { DALI_Commissioning.fbPart102Commands.bRecallMinLevel := TRUE; }
        Button (20,30 180x40), "Recall Max Level"
            OnMouseClick: execute { DALI_Commissioning.fbPart102Commands.bRecallMaxLevel := TRUE; }
        Button (260,180 111x40), "Down"
            OnMouseClick: execute { DALI_Commissioning.fbPart102Commands.bDown := TRUE; }
        Button (390,180 110x40), "Step Down"
            OnMouseClick: execute { DALI_Commissioning.fbPart102Commands.bStepDown := TRUE; }
        Button (260,130 240x40), "Step Down and Off"
            OnMouseClick: execute { DALI_Commissioning.fbPart102Commands.bStepDownAndOff := TRUE; }
        Button (660,30 80x40), "%d", text variable: DALI_Commissioning.fbPart102Commands.nScene
            OnMouseClick: write the text variable via Default, min 0, max 15, title "Insert scene number"
        Textfield (550,35 85x30), "Scene:"
        Button (560,80 180x40), "Go to Scene"
            OnMouseClick: execute { DALI_Commissioning.fbPart102Commands.bGotoScene := TRUE; }
        Button (260,80 240x40), "On and Step Up"
            OnMouseClick: execute { DALI_Commissioning.fbPart102Commands.bOnAndStepUp := TRUE; }
        Button (260,30 110x40), "Up"
            OnMouseClick: execute { DALI_Commissioning.fbPart102Commands.bUp := TRUE; }
        Button (390,30 110x40), "Step Up"
            OnMouseClick: execute { DALI_Commissioning.fbPart102Commands.bStepUp := TRUE; }
        Button (570,141 150x30), "Identify"
            OnMouseDown: execute { DALI_Commissioning.fbPart102Commands.bIdentify202 := TRUE; }
    GroupBox (420,60 370x230), "Status"
        Textfield (20,20 200x30), "Actual Level:"
        Textfield (20,60 200x30), "Control Gear Failure:"
        Textfield (231,20 50x30), "%s", text variable: DALI_Commissioning.fbPart102Commands.sActualLevel
        Textfield (230,60 50x30), "%s", text variable: DALI_Commissioning.fbPart102Commands.sControlGearFailure
        Textfield (20,100 200x30), "Lamp Failure:"
        Textfield (230,100 50x30), "%s", text variable: DALI_Commissioning.fbPart102Commands.sLampFailure
        Textfield (20,140 200x30), "Reset State:"
        Textfield (230,140 50x30), "%s", text variable: DALI_Commissioning.fbPart102Commands.sResetState
        Textfield (20,180 200x28), "Fade Running:"
        Textfield (230,180 50x30), "%s", text variable: DALI_Commissioning.fbPart102Commands.sFadeRunning
    GroupBox (10,60 390x230), "Address Type"
        Button (240,30 80x40), "%d", text variable: DALI_Commissioning.fbPart102Commands.nShortAddress
            OnMouseClick: write the text variable via Default, min 0, max 63, title "Insert Short Address"
            OnMouseClick: execute {  }
        RadioButton (20,20 190x200), variable: DALI_Commissioning.fbPart102Commands.eAddressType
            Areas[0]: Text=Short Address
            Areas[1]: Text=Group Address
            Areas[2]: Text=Broadcast
            Areas[3]: Text=Unaddressed
        Button (240,80 80x40), "%d", text variable: DALI_Commissioning.fbPart102Commands.nGroupAddress
            OnMouseClick: write the text variable via Default, min 0, max 15, title "Insert Group Address"
    Rectangle (720,0 70x15), "V%s", text variable: stLibVersion_Tc3_DALI_PLC_Commissioning_Tool.sVersion
    Group (10,5 170x40)
        Textfield (0,0 110x40), "DALI Line:"
        Button (90,0 80x40), "%d", text variable: GVL_Internal.nDALILine
            OnMouseClick: write the text variable via Default, min 1, max GVL_Internal.nNumberOfDALI_Lines, title "Choose line"
END_VISUALIZATION

// ---- Tc3_DALI_PLC_Commissioning_Tool/VISUs/Visu_DALICommissioning/Visu_Part102Groups.TcVIS
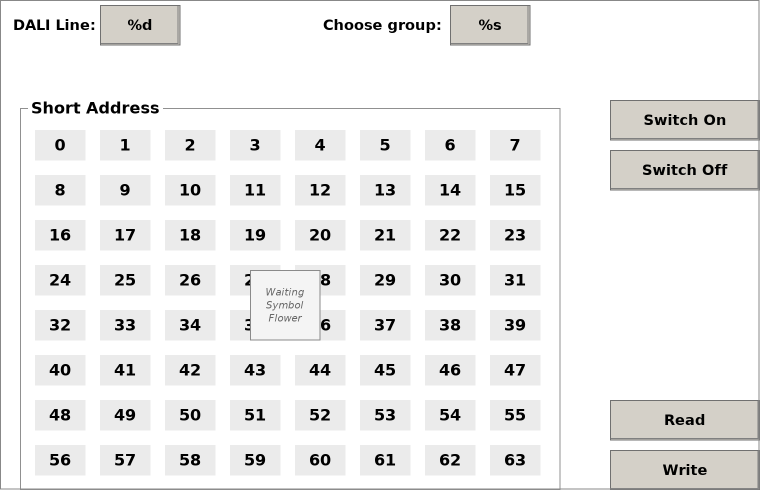
VISUALIZATION Visu_Part102Groups  // 760x490
    GroupBox (20,100 540x390), "Short Address"
        Textfield (15,30 50x30), "0", colour toggle: DALI_Commissioning.fbPart102Groups.aShowAlarmState[0] = TRUE, invisible if: DALI_Commissioning.fbPart102Groups.aActivateButton[0] = FALSE, input disabled if: DALI_Commissioning.fbPart102Groups.aActivateButton[0] = FALSE
            OnMouseClick: execute { DALI_Commissioning.fbPart102Groups.aButtonClick[0] := TRUE; }
        Textfield (80,30 50x30), "1", colour toggle: DALI_Commissioning.fbPart102Groups.aShowAlarmState[1] = TRUE, invisible if: DALI_Commissioning.fbPart102Groups.aActivateButton[1] = FALSE, input disabled if: DALI_Commissioning.fbPart102Groups.aActivateButton[1] = FALSE
            OnMouseClick: execute { DALI_Commissioning.fbPart102Groups.aButtonClick[1] := TRUE; }
        Textfield (145,30 50x30), "2", colour toggle: DALI_Commissioning.fbPart102Groups.aShowAlarmState[2] = TRUE, invisible if: DALI_Commissioning.fbPart102Groups.aActivateButton[2] = FALSE, input disabled if: DALI_Commissioning.fbPart102Groups.aActivateButton[2] = FALSE
            OnMouseClick: execute { DALI_Commissioning.fbPart102Groups.aButtonClick[2] := TRUE; }
        Textfield (210,30 50x30), "3", colour toggle: DALI_Commissioning.fbPart102Groups.aShowAlarmState[3] = TRUE, invisible if: DALI_Commissioning.fbPart102Groups.aActivateButton[3] = FALSE, input disabled if: DALI_Commissioning.fbPart102Groups.aActivateButton[3] = FALSE
            OnMouseClick: execute { DALI_Commissioning.fbPart102Groups.aButtonClick[3] := TRUE; }
        Textfield (275,30 50x30), "4", colour toggle: DALI_Commissioning.fbPart102Groups.aShowAlarmState[4] = TRUE, invisible if: DALI_Commissioning.fbPart102Groups.aActivateButton[4] = FALSE, input disabled if: DALI_Commissioning.fbPart102Groups.aActivateButton[4] = FALSE
            OnMouseClick: execute { DALI_Commissioning.fbPart102Groups.aButtonClick[4] := TRUE; }
        Textfield (340,30 50x30), "5", colour toggle: DALI_Commissioning.fbPart102Groups.aShowAlarmState[5] = TRUE, invisible if: DALI_Commissioning.fbPart102Groups.aActivateButton[5] = FALSE, input disabled if: DALI_Commissioning.fbPart102Groups.aActivateButton[5] = FALSE
            OnMouseClick: execute { DALI_Commissioning.fbPart102Groups.aButtonClick[5] := TRUE; }
        Textfield (405,30 50x30), "6", colour toggle: DALI_Commissioning.fbPart102Groups.aShowAlarmState[6] = TRUE, invisible if: DALI_Commissioning.fbPart102Groups.aActivateButton[6] = FALSE, input disabled if: DALI_Commissioning.fbPart102Groups.aActivateButton[6] = FALSE
            OnMouseClick: execute { DALI_Commissioning.fbPart102Groups.aButtonClick[6] := TRUE; }
        Textfield (470,30 50x30), "7", colour toggle: DALI_Commissioning.fbPart102Groups.aShowAlarmState[7] = TRUE, invisible if: DALI_Commissioning.fbPart102Groups.aActivateButton[7] = FALSE, input disabled if: DALI_Commissioning.fbPart102Groups.aActivateButton[7] = FALSE
            OnMouseClick: execute { DALI_Commissioning.fbPart102Groups.aButtonClick[7] := TRUE; }
        Textfield (15,75 50x30), "8", colour toggle: DALI_Commissioning.fbPart102Groups.aShowAlarmState[8] = TRUE, invisible if: DALI_Commissioning.fbPart102Groups.aActivateButton[8] = FALSE, input disabled if: DALI_Commissioning.fbPart102Groups.aActivateButton[8] = FALSE
            OnMouseClick: execute { DALI_Commissioning.fbPart102Groups.aButtonClick[8] := TRUE; }
        Textfield (80,75 50x30), "9", colour toggle: DALI_Commissioning.fbPart102Groups.aShowAlarmState[9] = TRUE, invisible if: DALI_Commissioning.fbPart102Groups.aActivateButton[9] = FALSE, input disabled if: DALI_Commissioning.fbPart102Groups.aActivateButton[9] = FALSE
            OnMouseClick: execute { DALI_Commissioning.fbPart102Groups.aButtonClick[9] := TRUE; }
        Textfield (145,75 50x30), "10", colour toggle: DALI_Commissioning.fbPart102Groups.aShowAlarmState[10] = TRUE, invisible if: DALI_Commissioning.fbPart102Groups.aActivateButton[10] = FALSE, input disabled if: DALI_Commissioning.fbPart102Groups.aActivateButton[10] = FALSE
            OnMouseClick: execute { DALI_Commissioning.fbPart102Groups.aButtonClick[10] := TRUE; }
        Textfield (210,75 50x30), "11", colour toggle: DALI_Commissioning.fbPart102Groups.aShowAlarmState[11] = TRUE, invisible if: DALI_Commissioning.fbPart102Groups.aActivateButton[11] = FALSE, input disabled if: DALI_Commissioning.fbPart102Groups.aActivateButton[11] = FALSE
            OnMouseClick: execute { DALI_Commissioning.fbPart102Groups.aButtonClick[11] := TRUE; }
        Textfield (275,75 50x30), "12", colour toggle: DALI_Commissioning.fbPart102Groups.aShowAlarmState[12] = TRUE, invisible if: DALI_Commissioning.fbPart102Groups.aActivateButton[12] = FALSE, input disabled if: DALI_Commissioning.fbPart102Groups.aActivateButton[12] = FALSE
            OnMouseClick: execute { DALI_Commissioning.fbPart102Groups.aButtonClick[12] := TRUE; }
        Textfield (340,75 50x30), "13", colour toggle: DALI_Commissioning.fbPart102Groups.aShowAlarmState[13] = TRUE, invisible if: DALI_Commissioning.fbPart102Groups.aActivateButton[13] = FALSE, input disabled if: DALI_Commissioning.fbPart102Groups.aActivateButton[13] = FALSE
            OnMouseClick: execute { DALI_Commissioning.fbPart102Groups.aButtonClick[13] := TRUE; }
        Textfield (405,75 50x30), "14", colour toggle: DALI_Commissioning.fbPart102Groups.aShowAlarmState[14] = TRUE, invisible if: DALI_Commissioning.fbPart102Groups.aActivateButton[14] = FALSE, input disabled if: DALI_Commissioning.fbPart102Groups.aActivateButton[14] = FALSE
            OnMouseClick: execute { DALI_Commissioning.fbPart102Groups.aButtonClick[14] := TRUE; }
        Textfield (470,75 50x30), "15", colour toggle: DALI_Commissioning.fbPart102Groups.aShowAlarmState[15] = TRUE, invisible if: DALI_Commissioning.fbPart102Groups.aActivateButton[15] = FALSE, input disabled if: DALI_Commissioning.fbPart102Groups.aActivateButton[15] = FALSE
            OnMouseClick: execute { DALI_Commissioning.fbPart102Groups.aButtonClick[15] := TRUE; }
        Textfield (15,120 50x30), "16", colour toggle: DALI_Commissioning.fbPart102Groups.aShowAlarmState[16] = TRUE, invisible if: DALI_Commissioning.fbPart102Groups.aActivateButton[16] = FALSE, input disabled if: DALI_Commissioning.fbPart102Groups.aActivateButton[16] = FALSE
            OnMouseClick: execute { DALI_Commissioning.fbPart102Groups.aButtonClick[16] := TRUE; }
        Textfield (80,120 50x30), "17", colour toggle: DALI_Commissioning.fbPart102Groups.aShowAlarmState[17] = TRUE, invisible if: DALI_Commissioning.fbPart102Groups.aActivateButton[17] = FALSE, input disabled if: DALI_Commissioning.fbPart102Groups.aActivateButton[17] = FALSE
            OnMouseClick: execute { DALI_Commissioning.fbPart102Groups.aButtonClick[17] := TRUE; }
        Textfield (145,120 50x30), "18", colour toggle: DALI_Commissioning.fbPart102Groups.aShowAlarmState[18] = TRUE, invisible if: DALI_Commissioning.fbPart102Groups.aActivateButton[18] = FALSE, input disabled if: DALI_Commissioning.fbPart102Groups.aActivateButton[18] = FALSE
            OnMouseClick: execute { DALI_Commissioning.fbPart102Groups.aButtonClick[18] := TRUE; }
        Textfield (210,120 50x30), "19", colour toggle: DALI_Commissioning.fbPart102Groups.aShowAlarmState[19] = TRUE, invisible if: DALI_Commissioning.fbPart102Groups.aActivateButton[19] = FALSE, input disabled if: DALI_Commissioning.fbPart102Groups.aActivateButton[19] = FALSE
            OnMouseClick: execute { DALI_Commissioning.fbPart102Groups.aButtonClick[19] := TRUE; }
        Textfield (275,120 50x30), "20", colour toggle: DALI_Commissioning.fbPart102Groups.aShowAlarmState[20] = TRUE, invisible if: DALI_Commissioning.fbPart102Groups.aActivateButton[20] = FALSE, input disabled if: DALI_Commissioning.fbPart102Groups.aActivateButton[20] = FALSE
            OnMouseClick: execute { DALI_Commissioning.fbPart102Groups.aButtonClick[20] := TRUE; }
        Textfield (340,120 50x30), "21", colour toggle: DALI_Commissioning.fbPart102Groups.aShowAlarmState[21] = TRUE, invisible if: DALI_Commissioning.fbPart102Groups.aActivateButton[21] = FALSE, input disabled if: DALI_Commissioning.fbPart102Groups.aActivateButton[21] = FALSE
            OnMouseClick: execute { DALI_Commissioning.fbPart102Groups.aButtonClick[21] := TRUE; }
        Textfield (405,120 50x30), "22", colour toggle: DALI_Commissioning.fbPart102Groups.aShowAlarmState[22] = TRUE, invisible if: DALI_Commissioning.fbPart102Groups.aActivateButton[22] = FALSE, input disabled if: DALI_Commissioning.fbPart102Groups.aActivateButton[22] = FALSE
            OnMouseClick: execute { DALI_Commissioning.fbPart102Groups.aButtonClick[22] := TRUE; }
        Textfield (470,120 50x30), "23", colour toggle: DALI_Commissioning.fbPart102Groups.aShowAlarmState[23] = TRUE, invisible if: DALI_Commissioning.fbPart102Groups.aActivateButton[23] = FALSE, input disabled if: DALI_Commissioning.fbPart102Groups.aActivateButton[23] = FALSE
            OnMouseClick: execute { DALI_Commissioning.fbPart102Groups.aButtonClick[23] := TRUE; }
        Textfield (15,165 50x30), "24", colour toggle: DALI_Commissioning.fbPart102Groups.aShowAlarmState[24] = TRUE, invisible if: DALI_Commissioning.fbPart102Groups.aDeviceGroupState[24] = 0, input disabled if: DALI_Commissioning.fbPart102Groups.aDeviceGroupState[24] = 0
            OnMouseClick: execute { DALI_Commissioning.fbPart102Groups.aButtonClick[24] := TRUE; }
        Textfield (80,165 50x30), "25", colour toggle: DALI_Commissioning.fbPart102Groups.aShowAlarmState[25] = TRUE, invisible if: DALI_Commissioning.fbPart102Groups.aActivateButton[25] = FALSE, input disabled if: DALI_Commissioning.fbPart102Groups.aActivateButton[25] = FALSE
            OnMouseClick: execute { DALI_Commissioning.fbPart102Groups.aButtonClick[25] := TRUE; }
        Textfield (145,165 50x30), "26", colour toggle: DALI_Commissioning.fbPart102Groups.aShowAlarmState[26] = TRUE, invisible if: DALI_Commissioning.fbPart102Groups.aActivateButton[26] = FALSE, input disabled if: DALI_Commissioning.fbPart102Groups.aActivateButton[26] = FALSE
            OnMouseClick: execute { DALI_Commissioning.fbPart102Groups.aButtonClick[26] := TRUE; }
        Textfield (210,165 50x30), "27", colour toggle: DALI_Commissioning.fbPart102Groups.aShowAlarmState[27] = TRUE, invisible if: DALI_Commissioning.fbPart102Groups.aActivateButton[27] = FALSE, input disabled if: DALI_Commissioning.fbPart102Groups.aActivateButton[27] = FALSE
            OnMouseClick: execute { DALI_Commissioning.fbPart102Groups.aButtonClick[27] := TRUE; }
        Textfield (275,165 50x30), "28", colour toggle: DALI_Commissioning.fbPart102Groups.aShowAlarmState[28] = TRUE, invisible if: DALI_Commissioning.fbPart102Groups.aActivateButton[28] = FALSE, input disabled if: DALI_Commissioning.fbPart102Groups.aActivateButton[28] = FALSE
            OnMouseClick: execute { DALI_Commissioning.fbPart102Groups.aButtonClick[28] := TRUE; }
        Textfield (340,165 50x30), "29", colour toggle: DALI_Commissioning.fbPart102Groups.aShowAlarmState[29] = TRUE, invisible if: DALI_Commissioning.fbPart102Groups.aActivateButton[29] = FALSE, input disabled if: DALI_Commissioning.fbPart102Groups.aActivateButton[29] = FALSE
            OnMouseClick: execute { DALI_Commissioning.fbPart102Groups.aButtonClick[29] := TRUE; }
        Textfield (405,165 50x30), "30", colour toggle: DALI_Commissioning.fbPart102Groups.aShowAlarmState[30] = TRUE, invisible if: DALI_Commissioning.fbPart102Groups.aActivateButton[30] = FALSE, input disabled if: DALI_Commissioning.fbPart102Groups.aActivateButton[30] = FALSE
            OnMouseClick: execute { DALI_Commissioning.fbPart102Groups.aButtonClick[30] := TRUE; }
        Textfield (470,165 50x30), "31", colour toggle: DALI_Commissioning.fbPart102Groups.aShowAlarmState[31] = TRUE, invisible if: DALI_Commissioning.fbPart102Groups.aActivateButton[31] = FALSE, input disabled if: DALI_Commissioning.fbPart102Groups.aActivateButton[31] = FALSE
            OnMouseClick: execute { DALI_Commissioning.fbPart102Groups.aButtonClick[31] := TRUE; }
        Textfield (15,210 50x30), "32", colour toggle: DALI_Commissioning.fbPart102Groups.aShowAlarmState[32] = TRUE, invisible if: DALI_Commissioning.fbPart102Groups.aActivateButton[32] = FALSE, input disabled if: DALI_Commissioning.fbPart102Groups.aActivateButton[32] = FALSE
            OnMouseClick: execute { DALI_Commissioning.fbPart102Groups.aButtonClick[32] := TRUE; }
        Textfield (80,210 50x30), "33", colour toggle: DALI_Commissioning.fbPart102Groups.aShowAlarmState[33] = TRUE, invisible if: DALI_Commissioning.fbPart102Groups.aActivateButton[33] = FALSE, input disabled if: DALI_Commissioning.fbPart102Groups.aActivateButton[33] = FALSE
            OnMouseClick: execute { DALI_Commissioning.fbPart102Groups.aButtonClick[33] := TRUE; }
        Textfield (145,210 50x30), "34", colour toggle: DALI_Commissioning.fbPart102Groups.aShowAlarmState[34] = TRUE, invisible if: DALI_Commissioning.fbPart102Groups.aActivateButton[34] = FALSE, input disabled if: DALI_Commissioning.fbPart102Groups.aActivateButton[34] = FALSE
            OnMouseClick: execute { DALI_Commissioning.fbPart102Groups.aButtonClick[34] := TRUE; }
        Textfield (210,210 50x30), "35", colour toggle: DALI_Commissioning.fbPart102Groups.aShowAlarmState[35] = TRUE, invisible if: DALI_Commissioning.fbPart102Groups.aActivateButton[35] = FALSE, input disabled if: DALI_Commissioning.fbPart102Groups.aActivateButton[35] = FALSE
            OnMouseClick: execute { DALI_Commissioning.fbPart102Groups.aButtonClick[35] := TRUE; }
        Textfield (275,210 50x30), "36", colour toggle: DALI_Commissioning.fbPart102Groups.aShowAlarmState[36] = TRUE, invisible if: DALI_Commissioning.fbPart102Groups.aActivateButton[36] = FALSE, input disabled if: DALI_Commissioning.fbPart102Groups.aActivateButton[36] = FALSE
            OnMouseClick: execute { DALI_Commissioning.fbPart102Groups.aButtonClick[36] := TRUE; }
        Textfield (340,210 50x30), "37", colour toggle: DALI_Commissioning.fbPart102Groups.aShowAlarmState[37] = TRUE, invisible if: DALI_Commissioning.fbPart102Groups.aActivateButton[37] = FALSE, input disabled if: DALI_Commissioning.fbPart102Groups.aActivateButton[37] = FALSE
            OnMouseClick: execute { DALI_Commissioning.fbPart102Groups.aButtonClick[37] := TRUE; }
        Textfield (405,210 50x30), "38", colour toggle: DALI_Commissioning.fbPart102Groups.aShowAlarmState[38] = TRUE, invisible if: DALI_Commissioning.fbPart102Groups.aActivateButton[38] = FALSE, input disabled if: DALI_Commissioning.fbPart102Groups.aActivateButton[38] = FALSE
            OnMouseClick: execute { DALI_Commissioning.fbPart102Groups.aButtonClick[38] := TRUE; }
        Textfield (470,210 50x30), "39", colour toggle: DALI_Commissioning.fbPart102Groups.aShowAlarmState[39] = TRUE, invisible if: DALI_Commissioning.fbPart102Groups.aActivateButton[39] = FALSE, input disabled if: DALI_Commissioning.fbPart102Groups.aActivateButton[39] = FALSE
            OnMouseClick: execute { DALI_Commissioning.fbPart102Groups.aButtonClick[39] := TRUE; }
        Textfield (15,255 50x30), "40", colour toggle: DALI_Commissioning.fbPart102Groups.aShowAlarmState[40] = TRUE, invisible if: DALI_Commissioning.fbPart102Groups.aActivateButton[40] = FALSE, input disabled if: DALI_Commissioning.fbPart102Groups.aActivateButton[40] = FALSE
            OnMouseClick: execute { DALI_Commissioning.fbPart102Groups.aButtonClick[40] := TRUE; }
        Textfield (80,255 50x30), "41", colour toggle: DALI_Commissioning.fbPart102Groups.aShowAlarmState[41] = TRUE, invisible if: DALI_Commissioning.fbPart102Groups.aActivateButton[41] = FALSE, input disabled if: DALI_Commissioning.fbPart102Groups.aActivateButton[41] = FALSE
            OnMouseClick: execute { DALI_Commissioning.fbPart102Groups.aButtonClick[41] := TRUE; }
        Textfield (145,255 50x30), "42", colour toggle: DALI_Commissioning.fbPart102Groups.aShowAlarmState[42] = TRUE, invisible if: DALI_Commissioning.fbPart102Groups.aActivateButton[42] = FALSE, input disabled if: DALI_Commissioning.fbPart102Groups.aActivateButton[42] = FALSE
            OnMouseClick: execute { DALI_Commissioning.fbPart102Groups.aButtonClick[42] := TRUE; }
        Textfield (210,255 50x30), "43", colour toggle: DALI_Commissioning.fbPart102Groups.aShowAlarmState[43] = TRUE, invisible if: DALI_Commissioning.fbPart102Groups.aActivateButton[43] = FALSE, input disabled if: DALI_Commissioning.fbPart102Groups.aActivateButton[43] = FALSE
            OnMouseClick: execute { DALI_Commissioning.fbPart102Groups.aButtonClick[43] := TRUE; }
        Textfield (275,255 50x30), "44", colour toggle: DALI_Commissioning.fbPart102Groups.aShowAlarmState[44] = TRUE, invisible if: DALI_Commissioning.fbPart102Groups.aActivateButton[44] = FALSE, input disabled if: DALI_Commissioning.fbPart102Groups.aActivateButton[44] = FALSE
            OnMouseClick: execute { DALI_Commissioning.fbPart102Groups.aButtonClick[44] := TRUE; }
        Textfield (340,255 50x30), "45", colour toggle: DALI_Commissioning.fbPart102Groups.aShowAlarmState[45] = TRUE, invisible if: DALI_Commissioning.fbPart102Groups.aActivateButton[45] = FALSE, input disabled if: DALI_Commissioning.fbPart102Groups.aActivateButton[45] = FALSE
            OnMouseClick: execute { DALI_Commissioning.fbPart102Groups.aButtonClick[45] := TRUE; }
        Textfield (405,255 50x30), "46", colour toggle: DALI_Commissioning.fbPart102Groups.aShowAlarmState[46] = TRUE, invisible if: DALI_Commissioning.fbPart102Groups.aActivateButton[46] = FALSE, input disabled if: DALI_Commissioning.fbPart102Groups.aActivateButton[46] = FALSE
            OnMouseClick: execute { DALI_Commissioning.fbPart102Groups.aButtonClick[46] := TRUE; }
        Textfield (470,255 50x30), "47", colour toggle: DALI_Commissioning.fbPart102Groups.aShowAlarmState[47] = TRUE, invisible if: DALI_Commissioning.fbPart102Groups.aActivateButton[47] = FALSE, input disabled if: DALI_Commissioning.fbPart102Groups.aActivateButton[47] = FALSE
            OnMouseClick: execute { DALI_Commissioning.fbPart102Groups.aButtonClick[47] := TRUE; }
        Textfield (15,300 50x30), "48", colour toggle: DALI_Commissioning.fbPart102Groups.aShowAlarmState[48] = TRUE, invisible if: DALI_Commissioning.fbPart102Groups.aActivateButton[48] = FALSE, input disabled if: DALI_Commissioning.fbPart102Groups.aActivateButton[48] = FALSE
            OnMouseClick: execute { DALI_Commissioning.fbPart102Groups.aButtonClick[48] := TRUE; }
        Textfield (80,300 50x30), "49", colour toggle: DALI_Commissioning.fbPart102Groups.aShowAlarmState[49] = TRUE, invisible if: DALI_Commissioning.fbPart102Groups.aActivateButton[49] = FALSE, input disabled if: DALI_Commissioning.fbPart102Groups.aActivateButton[49] = FALSE
            OnMouseClick: execute { DALI_Commissioning.fbPart102Groups.aButtonClick[49] := TRUE; }
        Textfield (145,300 50x30), "50", colour toggle: DALI_Commissioning.fbPart102Groups.aShowAlarmState[50] = TRUE, invisible if: DALI_Commissioning.fbPart102Groups.aActivateButton[50] = FALSE, input disabled if: DALI_Commissioning.fbPart102Groups.aActivateButton[50] = FALSE
            OnMouseClick: execute { DALI_Commissioning.fbPart102Groups.aButtonClick[50] := TRUE; }
        Textfield (210,300 50x30), "51", colour toggle: DALI_Commissioning.fbPart102Groups.aShowAlarmState[51] = TRUE, invisible if: DALI_Commissioning.fbPart102Groups.aActivateButton[51] = FALSE, input disabled if: DALI_Commissioning.fbPart102Groups.aActivateButton[51] = FALSE
            OnMouseClick: execute { DALI_Commissioning.fbPart102Groups.aButtonClick[51] := TRUE; }
        Textfield (275,300 50x30), "52", colour toggle: DALI_Commissioning.fbPart102Groups.aShowAlarmState[52] = TRUE, invisible if: DALI_Commissioning.fbPart102Groups.aActivateButton[52] = FALSE, input disabled if: DALI_Commissioning.fbPart102Groups.aActivateButton[52] = FALSE
            OnMouseClick: execute { DALI_Commissioning.fbPart102Groups.aButtonClick[52] := TRUE; }
        Textfield (340,300 50x30), "53", colour toggle: DALI_Commissioning.fbPart102Groups.aShowAlarmState[53] = TRUE, invisible if: DALI_Commissioning.fbPart102Groups.aActivateButton[53] = FALSE, input disabled if: DALI_Commissioning.fbPart102Groups.aActivateButton[53] = FALSE
            OnMouseClick: execute { DALI_Commissioning.fbPart102Groups.aButtonClick[53] := TRUE; }
        Textfield (405,300 50x30), "54", colour toggle: DALI_Commissioning.fbPart102Groups.aShowAlarmState[54] = TRUE, invisible if: DALI_Commissioning.fbPart102Groups.aActivateButton[54] = FALSE, input disabled if: DALI_Commissioning.fbPart102Groups.aActivateButton[54] = FALSE
            OnMouseClick: execute { DALI_Commissioning.fbPart102Groups.aButtonClick[54] := TRUE; }
        Textfield (470,300 50x30), "55", colour toggle: DALI_Commissioning.fbPart102Groups.aShowAlarmState[55] = TRUE, invisible if: DALI_Commissioning.fbPart102Groups.aActivateButton[55] = FALSE, input disabled if: DALI_Commissioning.fbPart102Groups.aActivateButton[55] = FALSE
            OnMouseClick: execute { DALI_Commissioning.fbPart102Groups.aButtonClick[55] := TRUE; }
        Textfield (15,345 50x30), "56", colour toggle: DALI_Commissioning.fbPart102Groups.aShowAlarmState[56] = TRUE, invisible if: DALI_Commissioning.fbPart102Groups.aActivateButton[56] = FALSE, input disabled if: DALI_Commissioning.fbPart102Groups.aActivateButton[56] = FALSE
            OnMouseClick: execute { DALI_Commissioning.fbPart102Groups.aButtonClick[56] := TRUE; }
        Textfield (80,345 50x30), "57", colour toggle: DALI_Commissioning.fbPart102Groups.aShowAlarmState[57] = TRUE, invisible if: DALI_Commissioning.fbPart102Groups.aActivateButton[57] = FALSE, input disabled if: DALI_Commissioning.fbPart102Groups.aActivateButton[57] = FALSE
            OnMouseClick: execute { DALI_Commissioning.fbPart102Groups.aButtonClick[56] := TRUE; }
        Textfield (145,345 50x30), "58", colour toggle: DALI_Commissioning.fbPart102Groups.aShowAlarmState[58] = TRUE, invisible if: DALI_Commissioning.fbPart102Groups.aActivateButton[58] = FALSE, input disabled if: DALI_Commissioning.fbPart102Groups.aActivateButton[58] = FALSE
            OnMouseClick: execute { DALI_Commissioning.fbPart102Groups.aButtonClick[58] := TRUE; }
        Textfield (210,345 50x30), "59", colour toggle: DALI_Commissioning.fbPart102Groups.aShowAlarmState[59] = TRUE, invisible if: DALI_Commissioning.fbPart102Groups.aActivateButton[59] = FALSE, input disabled if: DALI_Commissioning.fbPart102Groups.aActivateButton[59] = FALSE
            OnMouseClick: execute { DALI_Commissioning.fbPart102Groups.aButtonClick[59] := TRUE; }
        Textfield (275,345 50x30), "60", colour toggle: DALI_Commissioning.fbPart102Groups.aShowAlarmState[60] = TRUE, invisible if: DALI_Commissioning.fbPart102Groups.aActivateButton[60] = FALSE, input disabled if: DALI_Commissioning.fbPart102Groups.aActivateButton[60] = FALSE
            OnMouseClick: execute { DALI_Commissioning.fbPart102Groups.aButtonClick[60] := TRUE; }
        Textfield (340,345 50x30), "61", colour toggle: DALI_Commissioning.fbPart102Groups.aShowAlarmState[61] = TRUE, invisible if: DALI_Commissioning.fbPart102Groups.aActivateButton[61] = FALSE, input disabled if: DALI_Commissioning.fbPart102Groups.aActivateButton[61] = FALSE
            OnMouseClick: execute { DALI_Commissioning.fbPart102Groups.aButtonClick[61] := TRUE; }
        Textfield (405,345 50x30), "62", colour toggle: DALI_Commissioning.fbPart102Groups.aShowAlarmState[62] = TRUE, invisible if: DALI_Commissioning.fbPart102Groups.aActivateButton[62] = FALSE, input disabled if: DALI_Commissioning.fbPart102Groups.aActivateButton[62] = FALSE
            OnMouseClick: execute { DALI_Commissioning.fbPart102Groups.aButtonClick[62] := TRUE; }
        Textfield (470,345 50x30), "63", colour toggle: DALI_Commissioning.fbPart102Groups.aShowAlarmState[63] = TRUE, invisible if: DALI_Commissioning.fbPart102Groups.aActivateButton[63] = FALSE, input disabled if: DALI_Commissioning.fbPart102Groups.aActivateButton[63] = FALSE
            OnMouseClick: execute { DALI_Commissioning.fbPart102Groups.aButtonClick[63] := TRUE; }
        WaitingSymbolFlower (230,170 70x70), invisible if: DALI_Commissioning.fbPart102Groups.bHideWaitSymbol
    Button (610,400 150x40), "Read"
        OnMouseClick: execute { DALI_Commissioning.fbPart102Groups.bRead := TRUE; }
    Button (610,450 150x40), "Write"
        OnMouseClick: execute { DALI_Commissioning.fbPart102Groups.bWrite := TRUE; }
    Button (610,100 150x40), "Switch On"
        OnMouseClick: execute { DALI_Commissioning.fbPart102Groups.bSwitchOn := TRUE; }
    Button (610,150 150x40), "Switch Off"
        OnMouseClick: execute { DALI_Commissioning.fbPart102Groups.bSwitchOff := TRUE; }
    Group (320,5 210x40)
        Textfield (0,0 120x40), "Choose group:"
        Button (130,0 80x40), "%s", text variable: DALI_Commissioning.fbPart102Groups.nGroupAddress
            OnMouseClick: write the text variable via Default, min 0, max 15, title "Choose group"
    Group (10,5 170x40)
        Textfield (0,0 110x40), "DALI Line:"
        Button (90,0 80x40), "%d", text variable: GVL_Internal.nDALILine
            OnMouseClick: write the text variable via Default, min 1, max GVL_Internal.nNumberOfDALI_Lines, title "Choose line"
END_VISUALIZATION

// ---- Tc3_DALI_PLC_Commissioning_Tool/VISUs/Visu_DALICommissioning/Visu_Part102MemoryBank.TcVIS
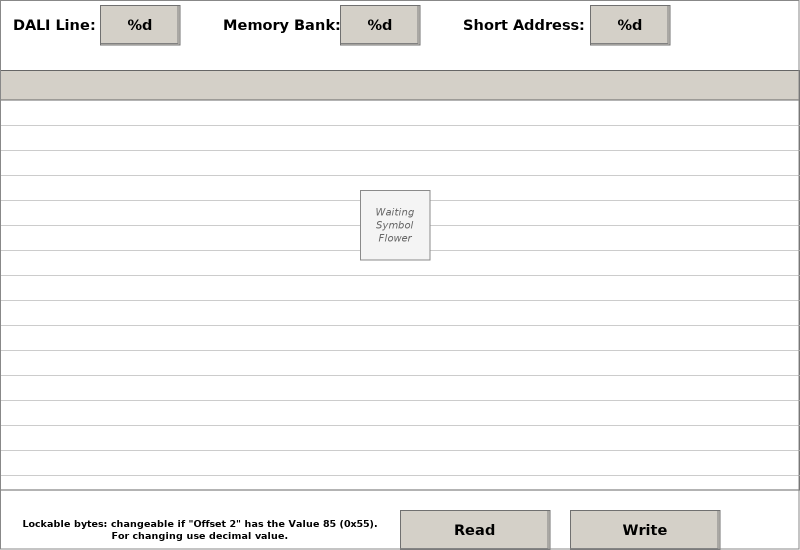
VISUALIZATION Visu_Part102MemoryBank  // 800x550
    Table (0,70 800x420), data array: DALI_Commissioning.fbPart102MemoryPages.aMemoryBank
        p1137915858: DALI_Commissioning.fbPart102MemoryPages.nOffset
        p3854506369: DALI_Commissioning.fbPart102MemoryPages.aMemoryBank[INDEX].sOffset
        p1892666644: DALI_Commissioning.fbPart102MemoryPages.aMemoryBank[INDEX].sName
        p338671338: DALI_Commissioning.fbPart102MemoryPages.aMemoryBank[INDEX].nValueDec
        p2170511999: DALI_Commissioning.fbPart102MemoryPages.aMemoryBank[INDEX].nValueHex
        p1755163831: Value Dec
        p4092479075: Value Hex
        Columns.Column.[0].Template: DALI_Commissioning.fbPart102MemoryPages.aNoValue[INDEX]
        Columns.Column.[1].Template: DALI_Commissioning.fbPart102MemoryPages.aNoValue[INDEX]
        Columns.Column.[2].Template: DALI_Commissioning.fbPart102MemoryPages.aNoValue[INDEX]; OnMouseClick: write the text variable via Default, min 0, max 255, title "Lockable variable decimal"
        Columns.Column.[3].Template: DALI_Commissioning.fbPart102MemoryPages.aNoValue[INDEX]; OnMouseClick: write the text variable via Default, title "Lockable variable hexadecimal"
    Button (400,510 150x40), "Read"
        OnMouseClick: execute { DALI_Commissioning.fbPart102MemoryPages.bRead := TRUE; }
    Button (570,510 150x40), "Write"
        OnMouseClick: execute { DALI_Commissioning.fbPart102MemoryPages.bWrite := TRUE; }
    Textfield (15,510 370x40), "Lockable bytes: changeable if "Offset 2" has the Value 85 (0x55). For changing use decimal value."
    WaitingSymbolFlower (360,190 70x70), invisible if: DALI_Commissioning.fbPart102MemoryPages.bHideWaitSymbol
    Textfield (460,5 130x40), "Short Address:"
    Button (590,5 80x40), "%d", text variable: DALI_Commissioning.fbPart102MemoryPages.nAddress
        OnMouseClick: write the text variable via Default, min 0, max 63, title "Insert Short Address"
    Textfield (220,5 120x40), "Memory Bank:"
    Button (340,5 80x40), "%d", text variable: DALI_Commissioning.fbPart102MemoryPages.nMemoryBank
        OnMouseClick: write the text variable via Default, min 0, max 255, title "Insert Memory Bank"
    Group (10,5 170x40)
        Textfield (0,0 110x40), "DALI Line:"
        Button (90,0 80x40), "%d", text variable: GVL_Internal.nDALILine
            OnMouseClick: write the text variable via Default, min 1, max GVL_Internal.nNumberOfDALI_Lines, title "Choose line"
END_VISUALIZATION

// ---- Tc3_DALI_PLC_Commissioning_Tool/VISUs/Visu_DALICommissioning/Visu_Part102Parameters.TcVIS
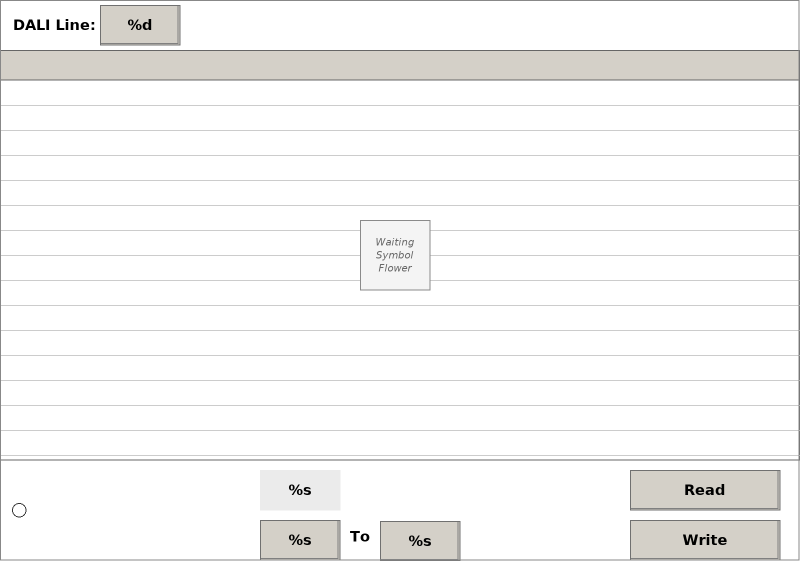
VISUALIZATION Visu_Part102Parameters  // 800x561
    Table (0,50 800x410), data array: DALI_Commissioning.fbPart102Parameters.aParameters
        p1137915858: DALI_Commissioning.fbPart102Parameters.nSelectedAddress
        p3854506369: DALI_Commissioning.fbPart102Parameters.aParameters[INDEX].nShortAddress
        p1892666644: DALI_Commissioning.fbPart102Parameters.aParameters[INDEX].nActualLevel
        p338671338: DALI_Commissioning.fbPart102Parameters.aParameters[INDEX].nMinLevel
        p2170511999: DALI_Commissioning.fbPart102Parameters.aParameters[INDEX].nMaxLevel
        p3723444502: DALI_Commissioning.fbPart102Parameters.aParameters[INDEX].eFadeRate
        p1218418051: DALI_Commissioning.fbPart102Parameters.aParameters[INDEX].eFadeTime
        p746581629: DALI_Commissioning.fbPart102Parameters.aParameters[INDEX].nPowerOnLevel
        p3104783080: DALI_Commissioning.fbPart102Parameters.aParameters[INDEX].nSystemFailureLevel
        p2501879983: DALI_Commissioning.fbPart102Parameters.aParameters[INDEX].nPhysicalMinimum
        p7306298: DALI_Commissioning.fbPart102Parameters.aParameters[INDEX].sDeviceTypes
        Columns.Column.[1].Template: OnMouseClick: write the text variable via Default, min 0, max 254, title "MinLevel"
        Columns.Column.[2].Template: OnMouseClick: write the text variable via Default, min 1, max 254, title "MaxLevel"
        Columns.Column.[3].Template: OnMouseClick: write the text variable via Default, min 0, max 254, title "FadeRate"
        Columns.Column.[4].Template: OnMouseClick: write the text variable via Default, min 1, max 15, title "Fade Rate"
        Columns.Column.[5].Template: OnMouseClick: write the text variable via Default, min 0, max 15, title "Fade Time"
        Columns.Column.[6].Template: OnMouseClick: write the text variable via Default, min 1, max 254, title "Power On Level"
        Columns.Column.[7].Template: OnMouseClick: write the text variable via Default, min 0, max 255, title "System Failure Level"
    RadioButton (10,460 254x100), variable: DALI_Commissioning.fbPart102Parameters.nAddressRange
        Areas[0]: Text=Single Short Address
        Areas[1]: Text=Short Address Range
    Textfield (335,521 50x31), "To"
    Button (630,470 150x40), "Read"
        OnMouseClick: execute { DALI_Commissioning.fbPart102Parameters.bRead := TRUE; }
    Button (630,520 150x40), "Write"
        OnMouseClick: execute { DALI_Commissioning.fbPart102Parameters.bWrite := TRUE; }
    Button (260,520 80x40), "%s", text variable: DALI_Commissioning.fbPart102Parameters.nStartAddress
        OnMouseClick: write the text variable via Default, min 0, max 63, title "Insert Short Address"
    Button (380,521 80x40), "%s", text variable: DALI_Commissioning.fbPart102Parameters.nEndAddress
        OnMouseClick: write the text variable via Default, min 0, max 63, title "Insert Short Address"
    Textfield (260,470 80x40), "%s", tooltip "Please select the desired Short Address in the table above.", text variable: DALI_Commissioning.fbPart102Parameters.nSelectedAddress
    WaitingSymbolFlower (360,220 70x70), invisible if: DALI_Commissioning.fbPart102Parameters.bHideWaitSymbol
    Group (10,5 170x40)
        Textfield (0,0 110x40), "DALI Line:"
        Button (90,0 80x40), "%d", text variable: GVL_Internal.nDALILine
            OnMouseClick: write the text variable via Default, min 1, max GVL_Internal.nNumberOfDALI_Lines, title "Choose line"
END_VISUALIZATION

